TYPE ST_SendDpCtrl :
STRUCT
	nRcvData				: WORD;
	nRcvSequenceNumber		: WORD;	
	nRcvCrc					: WORD;
END_STRUCT
END_TYPE

(* stored: Version 1.1.0.1, ProductVersion 3.1.4024.12
   DUT ST_SendDpCtrl: Id {fe6aaa6f-77d0-02dc-322b-7b238dc75ea4} *)
